TYPE T_Axis_Tx :
STRUCT
	CONTROL_WORD :UINT;
	TARGET_TORQUE:INT;
	MODE_OF_OPERATION:SINT:=4;
	MAX_MOTOR_SPEED : UDINT:=2000000;
END_STRUCT
END_TYPE

(* stored: Version 1.1.0.1, ProductVersion 3.1.4024.12
   DUT T_Axis_Tx: Id {515862d0-4a2e-4025-ab0f-5229bc8fe0ac} *)
